FUNCTION_BLOCK FB_CO2Sensor
VAR_INPUT
END_VAR
VAR_OUTPUT
END_VAR
VAR
	rCO2Value : REAL;
	iRange : INT := 32767;
	iVmax : INT := 10;
	iCorrespondenceFactor : INT := 1000;
END_VAR

rCO2Value := (INT_TO_REAL(MyGVL.iInput1)/iRange)*iVmax * iCorrespondenceFactor;

PROPERTY getCO2Value : REAL
GET
getCO2Value := rCO2Value;
END_GET
END_PROPERTY

END_FUNCTION_BLOCK

(* stored: Version 1.1.0.1, ProductVersion 3.1.4024.11
   POU FB_CO2Sensor: Id {61dcd89e-b219-4cf8-a2a7-d3d6a665d332}, SpecialFunc None
   Property getCO2Value: Id {4d729839-0a25-468b-a73b-6ded05b62662}
   Get Get: Id {8fbc6863-1d7a-4ff0-9640-75f589acb27c} *)
